{attribute 'qualified_only'}
VAR_GLOBAL CONSTANT
	// Mirrors Beckhoff's own Global_Version.stLibVersion_* pattern (see ST_LibVersion),
	// which only covers Tc2_*/Tc3_* library references, not custom ones like this one.
	// Kept in sync with <ProjectVersion> in HalfBROT.plcproj at release time.
	stVersion : ST_LibVersion := (
		iMajor := 0,
		iMinor := 4,
		iBuild := 0,
		iRevision := 0,
		nFlags := 1,
		sVersion := '0.4.0'
	);
END_VAR

(* stored: Version 1.1.0.1, ProductVersion 3.1.4024.15
   GVL GVL_Version: Id {6f45e4f1-e21a-4d69-b70c-b9b602163ca6} *)
